Omron CX-Programmer project NewProject (CX-Programmer 9.51)

# PLC my_first_project: CP1L L
; MyFirstProject

## Global symbols (name address type ; comment)
W0.04 BOOL  ; comment
W0.05 BOOL  ; comment

## Program NewProgram1 (cyclic task 0)
Local symbols
button_1 0.00 BOOL
out_1 100.00 BOOL
out_2 100.01 BOOL
out_3 100.02 BOOL

### Section Section1

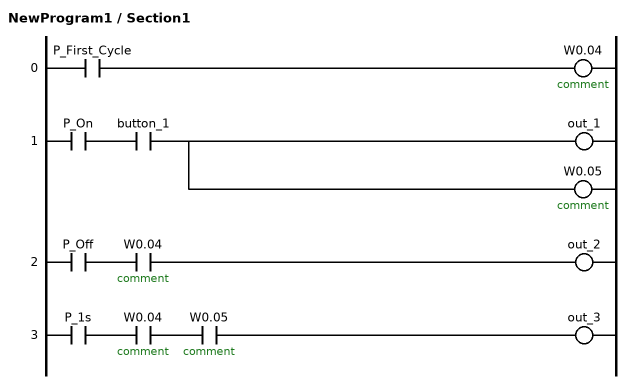
; rung 0
LD P_First_Cycle
OUT W0.04  ; comment
; rung 1
LD P_On
AND button_1
OUT out_1
OUT W0.05  ; comment
; rung 2
LD P_Off
AND W0.04  ; comment
OUT out_2
; rung 3
LD P_1s
AND W0.04  ; comment
AND W0.05  ; comment
OUT out_3

### Section END
; rung 0
END(001)